TYPE ST_OpenLoopControlData :
STRUCT
END_STRUCT
END_TYPE

(* stored: Version 1.1.0.1, ProductVersion 3.1.4024.12
   DUT ST_OpenLoopControlData: Id {ed4b6f74-8da2-4ccc-868f-9a3cac058366} *)
